      # point45 (the point 45 degrees along the path) (has no rxryrz data) (because if we do fixed angle circle move it wont use that anyways, it'l just use the angle from p1t)
      distup = cos(45 * pi/180) * (radius + cusharound)
      distover = sin(45 * pi/180) * (radius + cusharound)
      p45x = pcx + vecrx * distover + vecnx * -1 * cushout
      p45y = pcy + vecry * distover + vecny * -1 * cushout
      p45z = pcz + vecuz * distup
      point45 = p[p45x, p45y, p45z, 0,0,0]

      # point22 (22.5 degrees of angle)
      distup = cos(22.5 * pi/180) * (radius + cusharound)
      distover = sin(22.5 * pi/180) * (radius + cusharound)
      p22x = pcx + vecrx * distover + vecnx * -1 * cushout
      p22y = pcy + vecry * distover + vecny * -1 * cushout
      p22z = pcz + vecuz * distup
      point22 = p[p22x, p22y, p22z, 0,0,0]

      # return the points
      ret = struct(point1=point1, point2=point2, point3=point3, point4=point4, point1t=point1t, point45=point45, point22=point22)
      return ret

  end

  def make_pose_list(length):
      if length < 1:
          ret = []
          return ret
      end
      if length == 1:
          pose_list = [p[0, 0, 0, 0, 0, 0]]
          return pose_list
      end
      if length == 2:
          pose_list = [p[0, 0, 0, 0, 0, 0], p[0, 0, 0, 0, 0, 0]]
          return pose_list
      end
      if length == 3:
          pose_list = [p[0, 0, 0, 0, 0, 0], p[0, 0, 0, 0, 0, 0], p[0, 0, 0, 0, 0, 0]]
          return pose_list
      end
      if length == 4:
          pose_list = [p[0, 0, 0, 0, 0, 0], p[0, 0, 0, 0, 0, 0], p[0, 0, 0, 0, 0, 0], p[0, 0, 0, 0, 0, 0]]
          return pose_list
      end
      if length == 5:
          pose_list = [p[0, 0, 0, 0, 0, 0], p[0, 0, 0, 0, 0, 0], p[0, 0, 0, 0, 0, 0], p[0, 0, 0, 0, 0, 0], p[0, 0, 0, 0, 0, 0]]
          return pose_list
      end
      if length == 6:
          pose_list = [p[0, 0, 0, 0, 0, 0], p[0, 0, 0, 0, 0, 0], p[0, 0, 0, 0, 0, 0], p[0, 0, 0, 0, 0, 0], p[0, 0, 0, 0, 0, 0], p[0, 0, 0, 0, 0, 0]]
          return pose_list
      end
      if length == 7:
          pose_list = [p[0, 0, 0, 0, 0, 0], p[0, 0, 0, 0, 0, 0], p[0, 0, 0, 0, 0, 0], p[0, 0, 0, 0, 0, 0], p[0, 0, 0, 0, 0, 0], p[0, 0, 0, 0, 0, 0], p[0, 0, 0, 0, 0, 0]]
          return pose_list
      end
      if length == 8:
          pose_list = [p[0, 0, 0, 0, 0, 0], p[0, 0, 0, 0, 0, 0], p[0, 0, 0, 0, 0, 0], p[0, 0, 0, 0, 0, 0], p[0, 0, 0, 0, 0, 0], p[0, 0, 0, 0, 0, 0], p[0, 0, 0, 0, 0, 0], p[0, 0, 0, 0, 0, 0]]
          return pose_list
      end
      if length == 9:
          pose_list = [p[0, 0, 0, 0, 0, 0], p[0, 0, 0, 0, 0, 0], p[0, 0, 0, 0, 0, 0], p[0, 0, 0, 0, 0, 0], p[0, 0, 0, 0, 0, 0], p[0, 0, 0, 0, 0, 0], p[0, 0, 0, 0, 0, 0], p[0, 0, 0, 0, 0, 0], p[0, 0, 0, 0, 0, 0]]
          return pose_list
      end
      if length > 9:
          popuptext = "Program is only capable of storing 9 pegs at once. You selected more than 9. "
          # infinite loop
          while 1==1:
              popup(popuptext, title="Too Many Pegs",blocking=True)
          end
      end
  end

  # this function calculates the poses required on the weldpath for a specific teach pose for peg center.
  # call this function for every peg you want to weld.
  def main_calculate_peg(pose1):
      # constants
      peg_width = 2.05 # inches
      fixture_height = 1.5 # inches
      cushout = 0.006 # 5mm # the cushion out from the wall
      cusharound = 0.004 # 5mm # the cushion around the sleeve.
      delz = fixture_height *25.4/1000 - cushout
      rad = peg_width *1/2 * 25.4/1000 + cusharound

      # calculate angles
      # rxryrz1 (for point 1 (back side of peg)
      # start with gun facing up, shield tip pointing in x+ direction
      # rotate about y axis (y-) 135 degrees.
      # thats it. (for the other ones, then rotate 90 degrees about z axis from this spot
      m0 = get_rotation_matrix_from_description("y", -1, 225 * pi / 180)
      rxryrz1 = convert_matrix_to_axang(m0)
      rx1 = rxryrz1[0]
      ry1 = rxryrz1[1]
      rz1 = rxryrz1[2]

      # rxryrz2
      # second rotation is 90 degrees about z- axis
      m1 = get_rotation_matrix_from_description("z", -1, 90 * pi / 180)
      m2 = multiply_matrix(m1, m0)
      rxryrz2 = convert_matrix_to_axang(m2)
      rx2 = rxryrz2[0]
      ry2 = rxryrz2[1]
      rz2 = rxryrz2[2]

      # rxryrz3
      # second rotation is 180 degrees about z- axis
      m1 = get_rotation_matrix_from_description("z", -1, 180 * pi / 180)
      m2 = multiply_matrix(m1, m0)
      rxryrz3 = convert_matrix_to_axang(m2)
      rx3 = rxryrz3[0]
      ry3 = rxryrz3[1]
      rz3 = rxryrz3[2]

      # rxryrz4
      # second rotation is 270 degrees about z- axis
      m1 = get_rotation_matrix_from_description("z", -1, 270 * pi / 180)
      m2 = multiply_matrix(m1, m0)
      rxryrz4 = convert_matrix_to_axang(m2)
      rx4 = rxryrz4[0]
      ry4 = rxryrz4[1]
      rz4 = rxryrz4[2]

      # get points
      # get lift column height based on z value
      # if z is between +1 feet and -1 feet then go to 750
      # if z is greater than +1 feet but less than +4 feet, then go to 880
      # if z is greater than +4 feet, then error
      # if z is less than -1 feet, then go to 750 mm above z.

      # scrap that. new rules
      # go to 750 mm above z.
      # if that result is above 880, then go to 880.
      # that will work until we get problems

      z0 = pose1[2] # the teach point's z value (taken when lift column = 0)
      lczn = z0 + .750 # lift column z needed
      if lczn > .880:
          lczn = .880
      end
      liftcolumnzneeded = lczn * 1000 # set the z position
      zposerel = z0 - lczn # z pose relative = the teach point's z value at the new lift column position.

      pcenterx = pose1[0]
      pcentery = pose1[1]

      #points
      p1x = pcenterx - rad
      p1y = pcentery
      p1z = zposerel - delz

      p2x = pcenterx
      p2y = pcentery + rad
      p2z = zposerel - delz

      p3x = pcenterx + rad
      p3y = pcentery
      p3z = zposerel - delz

      p4x = pcenterx
      p4y = pcentery - rad
      p4z = zposerel - delz

      point1 = p[p1x, p1y, p1z, rx1, ry1, rz1]
      point2 = p[p2x, p2y, p2z, rx2, ry2, rz2]
      point3 = p[p3x, p3y, p3z, rx3, ry3, rz3]
      point4 = p[p4x, p4y, p4z, rx4, ry4, rz4]

      ret = struct(point1=point1, point2=point2, point3=point3, point4=point4, liftcolumnzneeded=liftcolumnzneeded)
      return ret



  end
  $ 137 "Set"
  set_tcp(p[1.4000000000000001E-4,-0.01751,0.284,0.0,0.0,0.0])
  $ 138 "Test_Teach_Peg()"
  Test_Teach_Peg()
  $ 139 "Set"
  set_tcp(p[1.4000000000000001E-4,-0.01751,0.284,0.0,0.0,0.0])
  $ 140 "kill threadId_Thread_1"
  kill threadId_Thread_1
  $ 142 "MoveL"
  $ 143 "Direction: Base Z+"
  global move_thread_flag_143=0
  thread move_thread_143():
    enter_critical
    move_thread_flag_143 = 1
    local towardsPos=calculate_point_to_move_towards(p[0.0,0.0,0.0,0.0,0.0,0.0], [0.0,0.0,1.0], 0.1)
    movel(towardsPos, a=1.2, v=0.25)
    move_thread_flag_143 = 2
    exit_critical
  end
  move_thread_flag_143 = 0
  move_thread_han_143 = run move_thread_143()
  while (True):
    sleep(1.0E-10)
    if (move_thread_flag_143 > 1):
      join move_thread_han_143
      $ 144 "Until (distance)"
      break
    end
    sync()
  end
  $ 145 "MoveJ"
  $ 146 "Waypoint_3" "breakAfter"
  movej(get_inverse_kin(Waypoint_3_p, qnear=Waypoint_3_q), a=1.3962634015954636, v=1.0471975511965976)
  $ 147 "Waypoint_40" "breakAfter"
  movej(get_inverse_kin(Waypoint_40_p, qnear=Waypoint_40_q), a=1.3962634015954636, v=1.0471975511965976)
  $ 148 "Set"
  set_tcp(p[-0.0095,-0.328,0.105,1.2092,-1.2092,1.2092])
  $ 149 "extrude knife"
  $ 150 "lch≔get_lift_column_height_condensed()"
  global lch=get_lift_column_height_condensed()
  $ 151 "If lch > 1"
  if (lch > 1):
    # begin: URCap Program Node
    #   Source: MachineLogic for Universal Robots, 3.1.7, Vention Inc.
    #   Type: MachineLogic for Universal Robots
    $ 152 "MachineLogic Homing"
    while isVentionMovementBusyMachineMotion1==True:
    sleep(0.05)
    end
    if(isVentionMovementBusyMachineMotion1 == False):
    isVentionMovementBusyMachineMotion1 = True
    socket_send_string("estop/status;", "MachineMotion1")
    temp_estop_var_vention = socket_read_string("MachineMotion1",timeout=15)
    while(temp_estop_var_vention=="estop/status true"):
    if temp_estop_var_vention=="estop/status true":
    sendStringWithTimeout("estop/systemreset/request","Ack estop/systemreset/request;","MachineMotion1")
    end
    socket_send_string("estop/status;", "MachineMotion1")
    temp_estop_var_vention = socket_read_string("MachineMotion1",timeout=15)
    if temp_estop_var_vention=="estop/status true":
    popup("MachineMotion in estop, make sure you have all emergency modules released manually. If you continue the system will try to reset MachineMotion automatically.",blocking=True)
    end
    end
    else:
    popup("resource is being used already: MachineMotion1")
    halt
    end
    isVentionMovementBusyMachineMotion1 = True
    sendString("im_home_axis_1", "MachineMotion im_home_axis_1 = completed", "MachineMotion1")
    isVentionMovementBusyMachineMotion1 = False
    sendString("SET im_set_encoder_pos_aux_1 0.000", "Ack", "MachineMotion1")
    isVentionMovementBusyMachineMotion1 = False
    sleep(0.03)
    # end: URCap Program Node
    $ 153 "extrude_knife3()"
    extrude_knife3()
    # begin: URCap Program Node
    #   Source: MachineLogic for Universal Robots, 3.1.7, Vention Inc.
    #   Type: MachineLogic for Universal Robots
    $ 154 "MachineLogic Move to Position"
    while isVentionMovementBusyMachineMotion1==True:
    sleep(0.05)
    end
    if(isVentionMovementBusyMachineMotion1 == False):
    isVentionMovementBusyMachineMotion1 = True
    socket_send_string("estop/status;", "MachineMotion1")
    temp_estop_var_vention = socket_read_string("MachineMotion1",timeout=15)
    while(temp_estop_var_vention=="estop/status true"):
    if temp_estop_var_vention=="estop/status true":
    sendStringWithTimeout("estop/systemreset/request","Ack estop/systemreset/request;","MachineMotion1")
    end
    socket_send_string("estop/status;", "MachineMotion1")
    temp_estop_var_vention = socket_read_string("MachineMotion1",timeout=15)
    if temp_estop_var_vention=="estop/status true":
    popup("MachineMotion in estop, make sure you have all emergency modules released manually. If you continue the system will try to reset MachineMotion automatically.",blocking=True)
    end
    end
    else:
    popup("resource is being used already: MachineMotion1")
    halt
    end
    sendString("SET speed_v2 3000000.000", "Ack", "MachineMotion1")
    sendString("SET acceleration_v2 50000.000", "Ack", "MachineMotion1")
    string_vention=intToString(lch*1000,"MachineMotion1")
    sendString("SET de_move_abs_1 "+string_vention, "Ack", "MachineMotion1")
    sendString("de_move_abs_exec", "Ack", "MachineMotion1")
    isVentionParallelMovementSendingScriptMachineMotion1 = False
    pollString("isMotionCompleted", "MachineMotion isMotionCompleted = true", "MachineMotion1")
    isVentionMovementBusyMachineMotion1 = False
    sleep(0.03)
    # end: URCap Program Node
  else:
    $ 155 "Else" "noBreak"
    $ 156 "extrude_knife3()"
    extrude_knife3()
  end
  $ 157 "dummy≔main_calculate_peg(poses_list[0])"
  global dummy=main_calculate_peg(poses_list[0])
  $ 158 "align_peg()"
  align_peg()
  $ 159 "pose_index≔0"
  global pose_index=0
  $ 160 "Loop pose_index < num_pegs"
  while (pose_index < num_pegs):
    $ 161 "peg_unwind()"
    peg_unwind()
    $ 162 "pose_cur≔poses_list[pose_index]"
    global pose_cur=poses_list[pose_index]
    $ 163 "pathturn≔main_calculate_peg(pose_cur)"
    global pathturn=main_calculate_peg(pose_cur)
    $ 164 "liftcolumnup"
    $ 165 "liftcolumnz≔liftcolumnzneeded"
    global liftcolumnz=liftcolumnzneeded
    # begin: URCap Program Node
    #   Source: MachineLogic for Universal Robots, 3.1.7, Vention Inc.
    #   Type: MachineLogic for Universal Robots
    $ 166 "MachineLogic Move to Position"
    while isVentionMovementBusyMachineMotion1==True:
    sleep(0.05)
    end
    if(isVentionMovementBusyMachineMotion1 == False):
    isVentionMovementBusyMachineMotion1 = True
    socket_send_string("estop/status;", "MachineMotion1")
    temp_estop_var_vention = socket_read_string("MachineMotion1",timeout=15)
    while(temp_estop_var_vention=="estop/status true"):
    if temp_estop_var_vention=="estop/status true":
    sendStringWithTimeout("estop/systemreset/request","Ack estop/systemreset/request;","MachineMotion1")
    end
    socket_send_string("estop/status;", "MachineMotion1")
    temp_estop_var_vention = socket_read_string("MachineMotion1",timeout=15)
    if temp_estop_var_vention=="estop/status true":
    popup("MachineMotion in estop, make sure you have all emergency modules released manually. If you continue the system will try to reset MachineMotion automatically.",blocking=True)
    end
    end
    else:
    popup("resource is being used already: MachineMotion1")
    halt
    end
    sendString("SET speed_v2 600000.000", "Ack", "MachineMotion1")
    sendString("SET acceleration_v2 50000.000", "Ack", "MachineMotion1")
    string_vention=intToString(liftcolumnz*1000,"MachineMotion1")
    sendString("SET de_move_abs_1 "+string_vention, "Ack", "MachineMotion1")
    sendString("de_move_abs_exec", "Ack", "MachineMotion1")
    isVentionParallelMovementSendingScriptMachineMotion1 = False
    pollString("isMotionCompleted", "MachineMotion isMotionCompleted = true", "MachineMotion1")
    isVentionMovementBusyMachineMotion1 = False
    sleep(0.03)
    # end: URCap Program Node
    $ 167 "weld_peg()"
    weld_peg()
    $ 168 "pose_index≔pose_index +1"
    global pose_index=pose_index +1
  end
  $ 171 "Set"
  set_tcp(p[-0.0095,-0.328,0.105,1.2092,-1.2092,1.2092])
  $ 172 "MoveJ"
  $ 173 "Waypoint_8" "breakAfter"
  movej(get_inverse_kin(Waypoint_8_p, qnear=Waypoint_8_q), a=1.3962634015954636, v=1.0471975511965976)
  $ 174 "Waypoint_9" "breakAfter"
  movej(get_inverse_kin(Waypoint_9_p, qnear=Waypoint_9_q), a=1.3962634015954636, v=1.0471975511965976)
  # begin: URCap Program Node
  #   Source: MachineLogic for Universal Robots, 3.1.7, Vention Inc.
  #   Type: MachineLogic for Universal Robots
  $ 175 "MachineLogic Homing"
  while isVentionMovementBusyMachineMotion1==True:
  sleep(0.05)
  end
  if(isVentionMovementBusyMachineMotion1 == False):
  isVentionMovementBusyMachineMotion1 = True
  socket_send_string("estop/status;", "MachineMotion1")
  temp_estop_var_vention = socket_read_string("MachineMotion1",timeout=15)
  while(temp_estop_var_vention=="estop/status true"):
  if temp_estop_var_vention=="estop/status true":
  sendStringWithTimeout("estop/systemreset/request","Ack estop/systemreset/request;","MachineMotion1")
  end
  socket_send_string("estop/status;", "MachineMotion1")
  temp_estop_var_vention = socket_read_string("MachineMotion1",timeout=15)
  if temp_estop_var_vention=="estop/status true":
  popup("MachineMotion in estop, make sure you have all emergency modules released manually. If you continue the system will try to reset MachineMotion automatically.",blocking=True)
  end
  end
  else:
  popup("resource is being used already: MachineMotion1")
  halt
  end
  isVentionMovementBusyMachineMotion1 = True
  sendString("im_home_axis_1", "MachineMotion im_home_axis_1 = completed", "MachineMotion1")
  isVentionMovementBusyMachineMotion1 = False
  sendString("SET im_set_encoder_pos_aux_1 0.000", "Ack", "MachineMotion1")
  isVentionMovementBusyMachineMotion1 = False
  sleep(0.03)
  # end: URCap Program Node
  $ 176 "Home"
  movej([-3.266929759358355, -1.2139462677784536, 1.5878387874396154, 1.1069165929565088, -0.0023738326664366483, -1.7891447305770605], a=1.3962634015954636, v=1.0471975511965976)
end
